TYPE DUT_stGetPLCData_Buffer :
STRUCT
	PLCData: STRING(DB.MAX_STRING_SIZE);
END_STRUCT
END_TYPE

(* stored: Version 1.1.0.1, ProductVersion 3.1.4024.15
   DUT DUT_stGetPLCData_Buffer: Id {ae9cab46-0c84-4f8c-ab98-e82001f72a4f} *)
